FUNCTION_BLOCK FB_GAM_PIP
VAR_INPUT
END_VAR
VAR_OUTPUT
END_VAR
VAR_IN_OUT
	stVolume : ST_Volume;
	stPip	:	ST_GAM_PIP;
END_VAR
VAR
	Pa 	: REAL;
	Va	: REAL;
END_VAR

(* Ion Pump Simulation
A. Pai 2017-1-27

The Ion Pump turns gas molecules into solid by using electroplating.

Therefore the Ion Pump takes gas molecules out of the system. 
We can treat that as if a small portion of gas mass is disappearing.

*)

IF stPip.xOn THEN

Pa := stVolume.rPressure;
Va := stVolume.rVolume;
// just reduce the pressure by 0.001%
stVolume.rPressure := Pa *(0.999);

END_IF

END_FUNCTION_BLOCK

(* stored: Version 1.1.0.1, ProductVersion 3.1.4020.12
   POU FB_GAM_PIP: Id {d08849ec-7e58-4f67-a60a-8aba2834a94e}, SpecialFunc None *)
